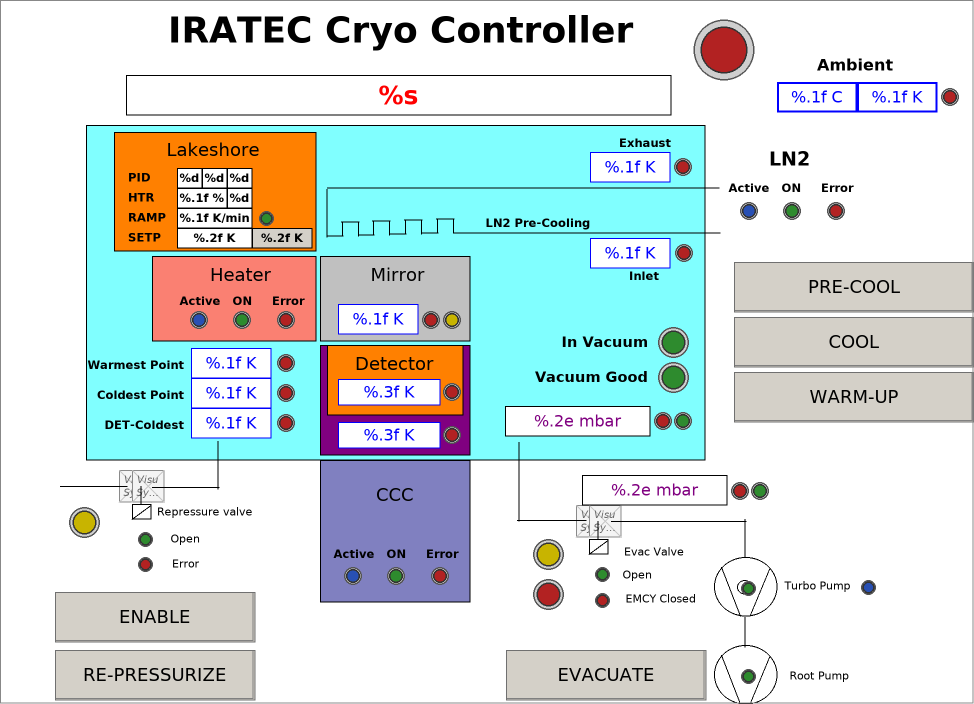
VISUALIZATION GUI_IRATEC  // 974x704
    RoundedRectangle (86,125 619x335)
    Group (327,188 393x50)
        Line (392,0) (0,0)
        Line (0,49) (0,1)
        Line (16,48) (0,48)
        Line (15,34) (15,48)
        Line (32,34) (14,34)
        Line (31,34) (31,48)
        Line (47,47) (31,47)
        Line (46,33) (46,47)
        Line (63,33) (45,33)
        Line (62,33) (62,47)
        Line (79,46) (63,46)
        Line (78,32) (78,46)
        Line (95,32) (77,32)
        Line (94,32) (94,46)
        Line (111,45) (95,45)
        Line (110,31) (110,45)
        Line (127,31) (109,31)
        Line (126,31) (126,45)
        Line (393,45) (126,45)
        Label (136,20 150x30), "LN2 Pre-Cooling"
    Group (714,557 63x59)
        Ellipse (0,0 63x59)
        Ellipse (23,23 15x14)
        Line (7,10) (26,59)
        Line (36,59) (56,11)
    Group (714,645 63x59)
        Ellipse (0,0 63x59)
        Line (7,10) (26,59)
        Line (36,59) (56,11)
    Line (745,647) (745,617)
    Image (576,505 32x32), image: VisuSymbols.Symbols.TriangleRight
    Group (589,505 32x49)
        Image (0,0 32x32), image: VisuSymbols.Symbols.TriangleLeft
        Rectangle (0,34 19x15)
        Line (0,49) (19,35)
        Line (9,34) (9,16)
    Line (745,557) (745,519)
    Line (611,521) (746,521)
    Line (517,520) (586,520)
    Line (519,521) (519,442)
    Rectangle (582,475 145x30), "%.2e mbar", text variable: MAIN.Cryo_Ctrl.Pressure_Evac.stat.lrPressure
    Rectangle (505,406 145x30), "%.2e mbar", text variable: MAIN.Cryo_Ctrl.Pressure_Cryo.stat.lrPressure
    Lamp1 (737,668 23x17), variable: MAIN.Cryo_Ctrl.EvacSys.stat.bRootPumpON, style: Lamp-Lamp1-Green
    Lamp1 (591,566 23x17), variable: MAIN.Cryo_Ctrl.EvacSys.stat.bValveOpen, style: Lamp-Lamp1-Green
    Image (119,470 32x32), image: VisuSymbols.Symbols.TriangleRight
    Group (132,470 32x49)
        Image (0,0 32x32), image: VisuSymbols.Symbols.TriangleLeft
        Rectangle (0,34 19x15)
        Line (0,49) (19,35)
        Line (9,34) (9,16)
    Lamp1 (134,531 23x17), variable: MAIN.Cryo_Ctrl.RepressValve.stat.bActON, style: Lamp-Lamp1-Green
    Line (218,489) (218,441)
    Line (152,487) (219,487)
    Line (60,486) (127,486)
    Label (130,497 150x30), "Repressure valve"
    Label (610,560 55x30), "Open"
    Lamp1 (656,360 35x35), variable: MAIN.Cryo_Ctrl.stat.bGoodVacuum, style: Lamp-Lamp1-Green
    Label (536,362 115x30), "Vacuum Good"
    Label (536,327 115x30), "In Vacuum"
    Lamp1 (656,325 35x35), variable: MAIN.Cryo_Ctrl.stat.bInVacuum, style: Lamp-Lamp1-Green
    Lamp1 (591,592 23x17), variable: MAIN.Cryo_Ctrl.EvacSys.stat.bEmergency, style: Lamp-Lamp1-Red
    Label (609,537 90x30), "Evac Valve"
    Label (614,584 94x30), "EMCY Closed"
    Lamp1 (737,580 23x17), variable: MAIN.Cryo_Ctrl.EvacSys.stat.bTurboPumpON, style: Lamp-Lamp1-Green
    Label (779,661 81x30), "Root Pump"
    Label (777,571 81x30), "Turbo Pump"
    Lamp1 (857,579 23x17), tooltip "Turbo Pump Ready", variable: MAIN.Cryo_Ctrl.EvacSys.stat.bTurboPump10min, style: Lamp-Lamp1-Blue
    Button (506,650 200x50), "EVACUATE", input disabled if: MAIN.Cryo_Ctrl.ctrl.bEnable_RepressSys=TRUE OR MAIN.Cryo_Ctrl.RepressValve.stat.bActON=TRUE
        toggle MAIN.Cryo_Ctrl.ctrl.bEnable_Evac
    Lamp1 (134,556 23x17), variable: MAIN.Cryo_Ctrl.RepressValve.stat.bError, style: Lamp-Lamp1-Red
    Label (158,524 55x30), "Open"
    Label (158,549 55x30), "Error"
    Button (55,592 200x50), "ENABLE", input disabled if: MAIN.Cryo_Ctrl.ctrl.bSafe_Repress=0
        toggle MAIN.Cryo_Ctrl.ctrl.bEnable_RepressSys
    Lamp1 (689,15 70x70), variable: MAIN.Cryo_Ctrl.stat.bError, invisible if: MAIN.Cryo_Ctrl.stat.bError = 0, style: Lamp-Lamp1-Red
    Rectangle (590,238 80x30), "%.1f K", text variable: MAIN.Cryo_Ctrl.Temp_LN2_Inlet.stat.lrTempK
    Rectangle (590,152 80x30), "%.1f K", text variable: MAIN.Cryo_Ctrl.Temp_LN2_Exhaust.stat.lrTempK
    Lamp1 (531,537 35x35), tooltip "If ON, system is enabled", variable: MAIN.Cryo_Ctrl.EvacSys.stat.bEnabled, style: Lamp-Lamp1-Yellow
    Lamp1 (67,505 35x35), tooltip "If ON, system is enabled", variable: MAIN.Cryo_Ctrl.ctrl.bEnable_RepressSys, style: Lamp-Lamp1-Yellow
    Group (716,144 150x77)
        Label (0,29 150x30), "Active ON Error"
        Lamp1 (23,57 20x20), variable: MAIN.Cryo_Ctrl.LN2.stat.bActive, style: Lamp-Lamp1-Blue
        Lamp1 (66,57 20x20), variable: MAIN.Cryo_Ctrl.LN2.stat.bActON, style: Lamp-Lamp1-Green
        Lamp1 (110,57 20x20), variable: MAIN.Cryo_Ctrl.LN2.stat.bError, style: Lamp-Lamp1-Red
        Label (36,0 75x30), "LN2"
    Lamp1 (531,577 35x35), tooltip "If ON, Evacuation System is in ERROR state.", variable: MAIN.Cryo_Ctrl.EvacSys.stat.bError, style: Lamp-Lamp1-Red
    Lamp1 (730,481 20x20), tooltip "Warning if reading is not valid", variable: NOT MAIN.Cryo_Ctrl.EvacSys.in_Pressure_Evac.bValid, style: Lamp-Lamp1-Red
    Group (320,460 151x142)
        Rectangle (0,0 150x142), "CCC"
        Lamp1 (23,106 20x20), tooltip "CCC Control is Enabled/Active", variable: MAIN.Cryo_Ctrl.CCC.stat.bActive, style: Lamp-Lamp1-Blue
        Lamp1 (66,106 20x20), tooltip "CCC is ON", variable: MAIN.Cryo_Ctrl.CCC.stat.bActON, style: Lamp-Lamp1-Green
        Lamp1 (110,106 20x20), variable: MAIN.Cryo_Ctrl.CCC.stat.bError, style: Lamp-Lamp1-Red
        Label (1,79 150x30), "Active ON Error"
    Label (602,128 86x30), "Exhaust"
    Label (601,261 86x30), "Inlet"
    Lamp1 (673,157 20x20), tooltip "Warning if reading is not valid", variable: NOT MAIN.Cryo_Ctrl.Temp_LN2_Exhaust.stat.bValid, style: Lamp-Lamp1-Red
    Lamp1 (674,243 20x20), tooltip "Warning if reading is not valid", variable: NOT MAIN.Cryo_Ctrl.Temp_LN2_Inlet.stat.bValid, style: Lamp-Lamp1-Red
    Lamp1 (653,411 20x20), tooltip "Warning if reading is not valid", variable: NOT MAIN.Cryo_Ctrl.Pressure_Cryo.stat.bValid, style: Lamp-Lamp1-Red
    Button (55,650 200x50), "RE-PRESSURIZE", input disabled if: MAIN.Cryo_Ctrl.ctrl.bEnable_RepressSys=0
        toggle MAIN.Cryo_Ctrl.ctrl.bEnable_RepressCtrl
    Button (734,262 240x50), "PRE-COOL", input disabled if: MAIN.Cryo_Ctrl.ctrl.bSafe_Precool = 0
        toggle MAIN.Cryo_Ctrl.ctrl.bEnable_Precool
    Button (734,317 240x50), "COOL", input disabled if: MAIN.Cryo_Ctrl.ctrl.bSafe_Cooling=0
        toggle MAIN.Cryo_Ctrl.ctrl.bEnable_Cool
    Button (734,372 240x50), "WARM-UP", input disabled if: MAIN.Cryo_Ctrl.ctrl.bSafe_Warmup=0
        toggle MAIN.Cryo_Ctrl.ctrl.bEnable_Warmup
    Label (152,5 498x50), "IRATEC Cryo Controller"
    Rectangle (126,75 545x40), "%s", text variable: MAIN.Cryo_Ctrl.stat.sState
    Group (152,256 165x85)
        Rectangle (0,0 164x85)
        Label (15,30 150x30), "Active ON Error"
        Lamp1 (37,54 20x20), tooltip "Heater Control is Enabled/Active", variable: MAIN.Cryo_Ctrl.Heater.stat.bActive, style: Lamp-Lamp1-Blue
        Lamp1 (80,54 20x20), tooltip "Heater is ON", variable: MAIN.Cryo_Ctrl.Heater.stat.bActON, style: Lamp-Lamp1-Green
        Lamp1 (124,54 20x20), variable: MAIN.Cryo_Ctrl.Heater.stat.bError, style: Lamp-Lamp1-Red
        Label (47,4 83x30), "Heater"
    Lamp1 (750,481 20x20), tooltip "Flag if reading is in sensor range", variable: MAIN.Cryo_Ctrl.EvacSys.in_Pressure_Evac.bInRange, style: Lamp-Lamp1-Green
    Lamp1 (673,411 20x20), tooltip "Flag if reading is in sensor range", variable: MAIN.Cryo_Ctrl.EvacSys.in_Pressure_Cryo.bInRange, style: Lamp-Lamp1-Green
    Label (92,380 95x30), "Coldest Point"
    Rectangle (191,378 80x30), "%.1f K", tooltip "Coldest point in the Cryostat", text variable: MAIN.Cryo_Ctrl.stat.lrLowestTempK
    Lamp1 (276,383 20x20), tooltip "Warning if reading is not valid", variable: NOT MAIN.Cryo_Ctrl.stat.bLowestTempValid, style: Lamp-Lamp1-Red
    Rectangle (191,408 80x30), "%.1f K", tooltip "Temperature difference between DET and the coldest point in the Cryostat", text variable: MAIN.Cryo_Ctrl.stat.lrDiffTempK
    Label (92,410 95x30), "DET-Coldest"
    Lamp1 (276,413 20x20), tooltip "Warning if reading is not valid", variable: NOT MAIN.Cryo_Ctrl.stat.bDiffTempValid, style: Lamp-Lamp1-Red
    Label (92,350 95x30), "Warmest Point"
    Rectangle (191,348 80x30), "%.1f K", tooltip "Warmest point in the Cryostat", text variable: MAIN.Cryo_Ctrl.stat.lrHighestTempK
    Lamp1 (276,353 20x20), tooltip "Warning if reading is not valid", variable: NOT MAIN.Cryo_Ctrl.stat.bHighestTempValid, style: Lamp-Lamp1-Red
    Rectangle (114,132 202x119)
    Label (160,135 106x30), "Lakeshore"
    Label (125,170 40x15), "PID"
    Label (125,190 40x15), "HTR"
    Label (125,210 40x15), "RAMP"
    Label (125,230 40x15), "SETP"
    Rectangle (177,168 25x20), "%d", text variable: MAIN.Cryo_Ctrl.Lakeshore.stat.nPID_P
    Rectangle (202,168 25x20), "%d", text variable: MAIN.Cryo_Ctrl.Lakeshore.stat.nPID_I
    Rectangle (227,168 25x20), "%d", text variable: MAIN.Cryo_Ctrl.Lakeshore.stat.nPID_D
    Rectangle (177,188 50x20), "%.1f %", tooltip "Heater Output [%]", text variable: MAIN.Cryo_Ctrl.Lakeshore.stat.lrHTR
    Rectangle (177,208 75x20), "%.1f K/min", tooltip "Heater Ramp Rate", text variable: MAIN.Cryo_Ctrl.Lakeshore.stat.lrRAMP_Rate
    Lamp1 (255,210 23x17), tooltip "Flag if Heater RAMP is On", variable: MAIN.Cryo_Ctrl.Lakeshore.stat.bRAMP_On, style: Lamp-Lamp1-Green
    Rectangle (177,228 75x20), "%.2f K", tooltip "SetPoint", text variable: MAIN.Cryo_Ctrl.Lakeshore.stat.lrSETP
    Rectangle (227,188 25x20), "%d", tooltip "Heater Range", text variable: MAIN.Cryo_Ctrl.Lakeshore.stat.nRANGE
    Group (320,256 150x85)
        Rectangle (0,0 150x85)
        Label (29,4 97x30), "Mirror"
        Rectangle (18,48 80x30), "%.1f K", text variable: MAIN.Cryo_Ctrl.Temp_Mirror.stat.lrTempK
        Lamp1 (101,54 20x20), tooltip "Warning if reading is not valid", variable: NOT MAIN.Cryo_Ctrl.Temp_Mirror.stat.bValid, style: Lamp-Lamp1-Red
        Lamp1 (122,54 20x20), tooltip "Warning if reading is underrange. PT100 cannot read below 73.15K (-200C).", variable: NOT MAIN.Cryo_Ctrl.Temp_Mirror.stat.bInRange, style: Lamp-Lamp1-Yellow
    Group (320,345 150x110)
        Rectangle (0,0 150x110)
        Rectangle (18,77 102x26), "%.3f K", tooltip "Heat Shield Temperature", text variable: MAIN.Cryo_Ctrl.Temp_HeatShield.stat.lrTempK
        Lamp1 (122,80 20x20), tooltip "Warning if reading is not valid", variable: NOT MAIN.Cryo_Ctrl.Temp_HeatShield.stat.bValid, style: Lamp-Lamp1-Red
    Group (327,345 136x70)
        Rectangle (0,0 136x70)
        Rectangle (11,34 102x26), "%.3f K", text variable: MAIN.Cryo_Ctrl.Temp_DET.stat.lrTempK
        Lamp1 (115,37 20x20), tooltip "Warning if reading is not valid", variable: NOT MAIN.Cryo_Ctrl.Temp_DET.stat.bValid, style: Lamp-Lamp1-Red
        Label (26,4 83x30), "Detector"
    Rectangle (252,228 60x20), "%.2f K", tooltip "Target SetPoint", text variable: MAIN.Cryo_Ctrl.Lakeshore.stat.lrSETP_Target
    Rectangle (857,82 80x30), "%.1f K", text variable: MAIN.Cryo_Ctrl.Temp_Ambient.stat.lrTempK
    Lamp1 (940,87 20x20), tooltip "Warning if reading is not valid", variable: NOT MAIN.Cryo_Ctrl.Temp_Ambient.stat.bValid, style: Lamp-Lamp1-Red
    Rectangle (777,82 80x30), "%.1f C", text variable: MAIN.Cryo_Ctrl.Temp_Ambient.stat.lrTempC
    Label (812,50 86x30), "Ambient"
END_VISUALIZATION

(* stored: Version 1.1.0.1, ProductVersion 3.1.4024.9
   Visu GUI_IRATEC: Id {ed460222-fdfd-4a68-81e4-07477aa6a355} *)
